(* IEC 61131-3 sources: 89152_FlorisHendrix_AfstudeerProject/89152_FlorisHendrix_ExamenProject/Stations/MachineControl/MachineControl/Class/GetOSVersion, 1 file *)

(* ---- GetOSVersion.st ---- *)
(*!
<Class
	Name               = "GetOSVersion"
	Revision           = "1.2"
	RealtimeTask       = "false"
	CyclicTask         = "false"
	BackgroundTask     = "false"
	Sigmatek           = "false"
	OSInterface        = "false"
	HighPriority       = "false"
	Automatic          = "false"
	UpdateMode         = "Prescan"
	SharedCommandTable = "true"
	Objectsize         = "(510,180)"
	Comment            = "class to read the OS version and write it to a string object ">
	<Channels>
		<Server Name="ClassSvr" Visualized="false" Initialize="false" WriteProtected="false" Retentive="false" Comment="class server"/>
		<Client Name="cAsciiBin" Required="true" Internal="false" Comment="object channel to a ASCII_BIN object &#13;&#10;to convert the os version from Bin to ASCII "/>
		<Client Name="cOSVersion" Required="true" Internal="false" Comment="object channel to a string object &#13;&#10;to write os version on stringram"/>
	</Channels>
	<Dependencies>
		<Files>
			<File Path=".\Class\GetOSVersion\GetOSVersion_de.pdf"/>
			<File Path=".\Class\GetOSVersion\GetOSVersion_en.pdf"/>
		</Files>
	</Dependencies>
	<RevDoku>
		<Owner Company="Sigmatek"/>
		<Dokumentation Revision="1.2" Date="2017-08-02" Author="FurLuk" Company="Sigmatek" Description="changed formatting"/>
		<Dokumentation Revision="1.1" Date="2016-10-10" Author="HubChr" Company="Sigmatek" Description="Added documentation pdfs."/>
		<Dokumentation Revision="1.0" Date="2015-09-22" Company="Sigmatek" Description="Creation."/>
	</RevDoku>
</Class>
*)
GetOSVersion : CLASS
  //Servers:
	ClassSvr 	: SvrChCmd_DINT;
  //Clients:
	cOSVersion 	: CltChCmd_String;
	cAsciiBin 	: CltChCmd_ASCII_BIN;
  //Variables:
		String : ARRAY [0..20] OF CHAR;

		Temp : ARRAY [0..20] OF CHAR;

  //Functions:

	FUNCTION VIRTUAL GLOBAL Init;

	FUNCTION GLOBAL OSVersion;

	FUNCTION VIRTUAL GLOBAL ClassSvr::Write
		VAR_INPUT
			input (EAX) 	: DINT;
		END_VAR
		VAR_OUTPUT
			result (EAX) 	: DINT;
		END_VAR;
  //Tables:
	FUNCTION @STD
		VAR_OUTPUT
			ret_code	: CONFSTATES;
		END_VAR;
	FUNCTION GLOBAL TAB @CT_;
END_CLASS;

#pragma usingLtd ASCII_BIN
#pragma usingLtd String

FUNCTION VIRTUAL GLOBAL GetOSVersion::Init

  if _firstscan then
    OSVersion();
  end_if;

END_FUNCTION

FUNCTION VIRTUAL GLOBAL GetOSVersion::ClassSvr::Write
	VAR_INPUT
		input (EAX) 	: DINT;
	END_VAR
	VAR_OUTPUT
		result (EAX) 	: DINT;
	END_VAR

	ClassSvr := input;
  OSVersion();
 	result := ClassSvr;

END_FUNCTION

FUNCTION GLOBAL GetOSVersion::OSVersion

  if (_rtosversion AND 16#F000) <> 0 then

    cAsciiBin.Bin2Ascii(#String$CHAR, ((_rtosversion AND 16#F000) SHR 12)$DINT, 16#0102);

    cAsciiBin.Bin2Ascii(#Temp$CHAR, ((_rtosversion AND 16#0F00) SHR 8)$DINT, 16#0222);
    _strcat(#String$CHAR, #Temp$CHAR);

    cAsciiBin.Bin2Ascii(#Temp$CHAR, (_rtosversion AND 16#FF)$DINT,16#0033);
    _strcat(#String$CHAR, #Temp$CHAR);

   // write os version on stringram
   cOSVersion.WriteDataOff(21,0,#String$USINT);

  end_if;

END_FUNCTION
